{attribute 'qualified_only'}
{attribute 'strict'}
TYPE E_CRYO_BIN_ACT_CMD :
(
	NONE	:= 0,
	OFF 	:= 1,
	ON		:= 2
);
END_TYPE

(* stored: Version 1.1.0.1, ProductVersion 3.1.4024.9
   DUT E_CRYO_BIN_ACT_CMD: Id {ad374623-bb86-471f-a131-3c0e9e1b8f68} *)
